// TIA Portal V20 export
TYPE "typeEm7CommandsJobInterface"
// stored: Access Published, Namespace Unit1
   STRUCT
      reqManPpUnloading { ExternalWritable := 'False'} : Bool;
      reqVisionInspection { ExternalWritable := 'False'} : Bool;
   END_STRUCT;
END_TYPE
